Fanuc KAREL source: kt00012.KL

-- PROVISIONAL review KL for V770-1; original PC SHA256 1b50d1c6a578d27e85e6367ebd30428245432dfff86cbe0926bd059deca0dee5
-- Incomplete behavior may be omitted. Consult companion uncertainty JSON. Do not deploy.
PROGRAM KT00012
%NOLOCKGROUP
VAR
  R1 : REAL
  R2 : REAL
  OUT : REAL
BEGIN
  -- UNRESOLVED_PC offsets 5-16; opcodes 2E,23
  -- UNRESOLVED_PC offsets 21-32; opcodes 2E,23
  -- UNRESOLVED_PC offsets 37-48; opcodes 2E,23
  -- UNRESOLVED_PC offsets 53-64; opcodes 2E,23
  -- UNRESOLVED_PC offsets 69-88; opcodes 21,21,69,23
  -- UNRESOLVED_PC offsets 93-97; opcodes 7F
END KT00012
